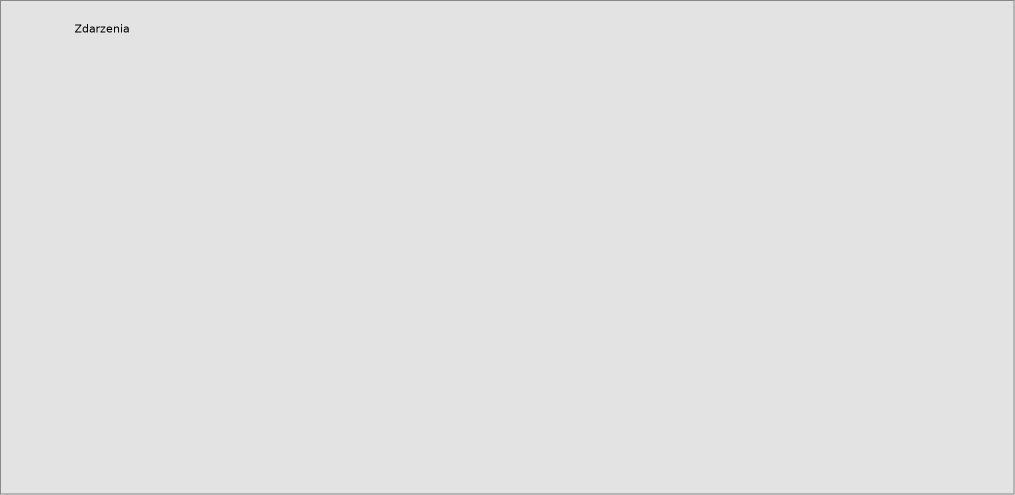
VISUALIZATION F_03_Events  // 1015x495
VAR_IN_OUT
	stScreenData	: ST_MCHMIPrepareScreen_03_XX;
	
END_VAR
    Label (27,14 150x30), "Zdarzenia"
END_VISUALIZATION

(* stored: Version 1.1.0.1
   Visu F_03_Events: Id {e1c2cb19-491b-0735-1b9c-f392d18e0493} *)
